// Mitsubishi GX Works2 project: CODIGO CLP   PLC: FX3U/FX3UC
// Configuração Modbus RTU

PROGRAM MAIN
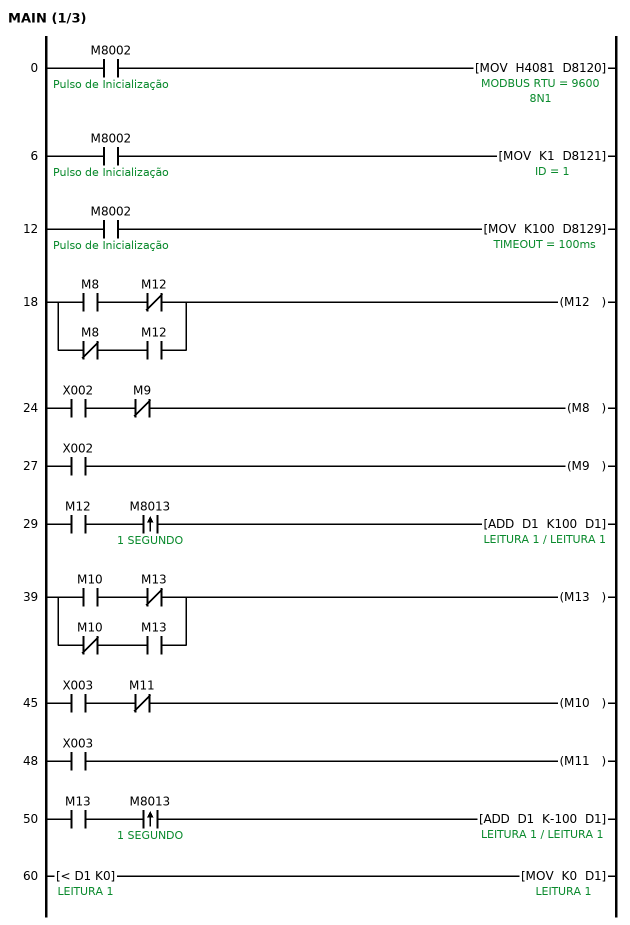
0     LD      M8002  ; Pulso de Inicialização
      MOV     H4081 D8120  ; MODBUS RTU = 9600 8N1
6     LD      M8002  ; Pulso de Inicialização
      MOV     K1 D8121  ; ID = 1
12    LD      M8002  ; Pulso de Inicialização
      MOV     K100 D8129  ; TIMEOUT = 100ms
18    LD      M8
      ANI     M12
      LDI     M8
      AND     M12
      ORB
      OUT     M12
24    LD      X002
      ANI     M9
      OUT     M8
27    LD      X002
      OUT     M9
29    LD      M12
      ANDP    M8013  ; 1 SEGUNDO
      ADD     D1 K100 D1  ; LEITURA 1
39    LD      M10
      ANI     M13
      LDI     M10
      AND     M13
      ORB
      OUT     M13
45    LD      X003
      ANI     M11
      OUT     M10
48    LD      X003
      OUT     M11
50    LD      M13
      ANDP    M8013  ; 1 SEGUNDO
      ADD     D1 K-100 D1
60    LD<     D1 K0  ; LEITURA 1
      MOV     K0 D1
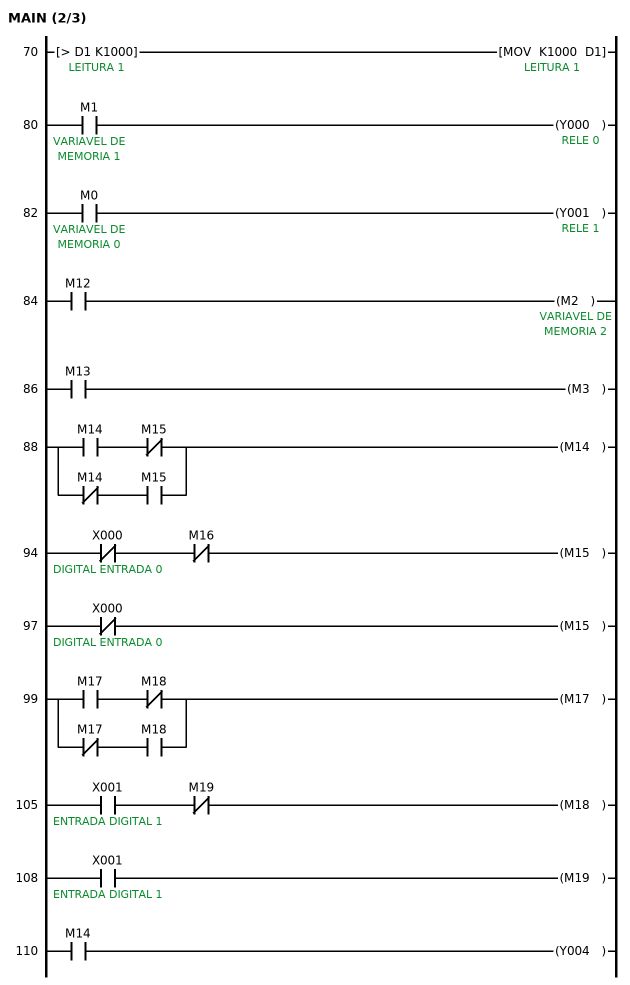
70    LD>     D1 K1000  ; LEITURA 1
      MOV     K1000 D1
80    LD      M1  ; VARIAVEL DE MEMORIA 1
      OUT     Y000  ; RELE 0
82    LD      M0  ; VARIAVEL DE MEMORIA 0
      OUT     Y001  ; RELE 1
84    LD      M12
      OUT     M2  ; VARIAVEL DE MEMORIA 2
86    LD      M13
      OUT     M3
88    LD      M14
      ANI     M15
      LDI     M14
      AND     M15
      ORB
      OUT     M14
94    LDI     X000  ; DIGITAL ENTRADA 0
      ANI     M16
      OUT     M15
97    LDI     X000  ; DIGITAL ENTRADA 0
      OUT     M15
99    LD      M17
      ANI     M18
      LDI     M17
      AND     M18
      ORB
      OUT     M17
105   LD      X001  ; ENTRADA DIGITAL 1
      ANI     M19
      OUT     M18
108   LD      X001  ; ENTRADA DIGITAL 1
      OUT     M19
110   LD      M14
      OUT     Y004
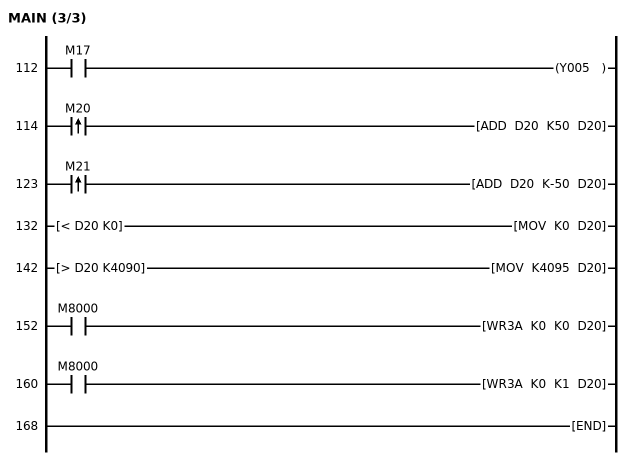
112   LD      M17
      OUT     Y005
114   LDP     M20
      ADD     D20 K50 D20
123   LDP     M21
      ADD     D20 K-50 D20
132   LD<     D20 K0
      MOV     K0 D20
142   LD>     D20 K4090
      MOV     K4095 D20
152   LD      M8000
      WR3A    K0 K0 D20
160   LD      M8000
      WR3A    K0 K1 D20
168   END
END_PROGRAM

// device comments not shown above
Y002  ; RELE 2
D0  ; REGISTRO 0
D2  ; ENCHE O TANQUE
D3  ; ESVAZIA O TANQUE
